(* IEC 61131-3 sources: echidna/examples, 8 files *)

(* ---- fb.il ---- *)
(*
    This is a non-functional instruction list application which is the subject
    of further echidna virtual machine development.
*)

function_block toggle
var_input run: bool; end_var
var_input cycle: time; end_var
var_output q: bool; end_var

ld run
st q

end_function_block

program test
var blink: toggle; end_var
var count: uint := 0; end_var

cal blink(
    run := true,
    cycle := t#500ms
)
dbg blink.q

add count, 1
st count
eq 5
retcn
_exit

end_program

configuration config1

task task1 (interval := t#1s, priority := 1);
program program1 with task1: test;

end_configuration

(* ---- blink.il ---- *)
(* Incrementally toggling 0/1 output driven by ton/ton/f_trig/r_trig *)

program test
var inp: bool; end_var
var cycle: time := t#500ms; end_var
var t1, t2: ton; end_var
var redge: r_trig; end_var
var fedge: f_trig; end_var

ldn t2.q
st inp
cal t1(
    in := inp,
    pt := cycle
)
cal t2(
    in := t1.q,
    pt := cycle
)

cal redge(
    clk := t1.q
)
ld redge.q
jmpcn down
dbg 1   (* Print 1 *)
down: cal fedge(
    clk := t1.q
)
ld fedge.q
retcn
dbg 0   (* Print 0 *)

end_program

configuration config1
task task1 (interval := t#10ms, priority := 1);
program program1 with task1: test;
end_configuration

(* ---- ctu.il ---- *)
program test
var count: ctu; end_var
var maxval: sint := 10; end_var

cal count(
    cu := true,
    pv := maxval,
    r := count.q
)
dbg count.q

end_program

configuration config1

task task1 (interval := t#100ms, priority := 1);
program program1 with task1: test;

end_configuration

(* ---- factorial.il ---- *)
function fact: udint
var_input inp: udint; end_var
var_output out: udint; end_var
var local: udint; end_var

ld inp
ge 1
jmpc nonzero
ld 1
ret
nonzero: ld inp
sub 1
st local
fact local
mul inp
st out
ret

end_function

program test
var cycle, result: udint := 0; end_var

fact cycle
st result
dbg cycle, result

add cycle, 1
st cycle
le 10  (* Limit execution to 11 cycles *)
retc
_exit

end_program

configuration config1
task task1 (interval := t#50ms, priority := 1);
program program1 with task1: test;
end_configuration

(* ---- rpiface-updown.il ---- *)
program test
var val: byte := 1; end_var
var dir: bool := true; end_var

piface_write val

ld dir
jmpcn rshift

lshift: shl val, 1
st val
eq 128
r dir
ret

rshift: shr val, 1
st val
eq 1
s dir
ret

end_program

configuration config1
task task1 (interval := t#80ms, priority := 1);
program program1 with task1: test;
end_configuration

(* ---- rpiface.il ---- *)
program test
var inp, val: byte := 1; end_var
var res: bool; end_var

piface_read
st inp
eq 0
jmpc roll

ld inp
and val
eq val
jmpcn roll
piface_write inp        (* Mirror inputs if asserted *)
ret

roll: piface_write val  (* Otherwise roll outputs *)
rol val, 1
st val

end_program

configuration config1
task task1 (interval := t#100ms, priority := 1);
program program1 with task1: test;
end_configuration

(* ---- rtc.il ---- *)
(* Output current time once per second *)

program test
var clock: rtc; end_var

cal clock
dbg clock.cdt

end_program

configuration config1
task task1 (interval := t#1s, priority := 1);
program program1 with task1: test;
end_configuration

(* ---- sine.il ---- *)
PROGRAM prog1
VAR cycle: UINT := 0; END_VAR
VAR bias: REAL := 0; END_VAR
VAR magnitude: REAL := 100; END_VAR
VAR samples: REAL := 200; END_VAR
VAR value: REAL; END_VAR

LD cycle
ADD 1
ST cycle
uint_to_real cycle
MUL 6.2831854 (* 2pi *)
DIV samples
ST value
sin value
MUL magnitude
ADD bias
ST value
dbg value

END_PROGRAM

CONFIGURATION config1
TASK task1 (INTERVAL := t#50ms, PRIORITY := 1);
PROGRAM program1 WITH task1: prog1;
END_CONFIGURATION
